Yaskawa INFORM job: Test.jbi

/JOB
//NAME TEST
//POS
///NPOS 0,0,0,0,0,0
//INST
///DATE 2007/07/24 10:22
///ATTR SC,RW
NOP
'TESTJOB
SET B000 1
END
